FUNCTION_BLOCK DataSelector (* Basic Function Block Type *)
  (* Standard: 61499-2 *)
  (* Version 0.0, 9/17/2024, midxav, Template *)
  PACKAGE Main;
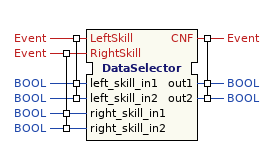
  EVENT_INPUT
    LeftSkill WITH left_skill_in1, left_skill_in2; (* Normal Execution Request *)
    RightSkill WITH right_skill_in1, right_skill_in2;
  END_EVENT
  EVENT_OUTPUT
    CNF WITH out1, out2; (* Execution Confirmation *)
  END_EVENT
  VAR_INPUT
    left_skill_in1 : BOOL; (* Input event qualifier *)
    left_skill_in2 : BOOL;
    right_skill_in1 : BOOL;
    right_skill_in2 : BOOL;
  END_VAR
  VAR_OUTPUT
    out1 : BOOL; (* Output event qualifier *)
    out2 : BOOL;
  END_VAR
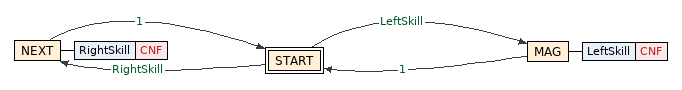
  EC_STATES
    START; (* Initial State *)
    MAG : LeftSkill -> CNF;
    NEXT : RightSkill -> CNF;
  END_STATES
  EC_TRANSITIONS
    START TO MAG := LeftSkill;
    MAG TO START := 1;
    START TO NEXT := RightSkill;
    NEXT TO START := 1;
  END_TRANSITIONS
  ALGORITHM INIT IN ST: (* Initialization algorithm *)
;
  END_ALGORITHM
  ALGORITHM REQ IN ST: (* Normally executed algorithm *)
;
  END_ALGORITHM
  ALGORITHM LeftSkill IN ST:
out1:=left_skill_in1;
out2:=left_skill_in2;
  END_ALGORITHM
  ALGORITHM RightSkill IN ST:
out1:=right_skill_in1;
out2:=right_skill_in2;
  END_ALGORITHM
END_FUNCTION_BLOCK
